FUNCTION_BLOCK AI_1_Module
VAR
	{attribute addProperty Name  "1"}
	iCHANNEL_1 : AI_Channel;
	{attribute addProperty Name  "WcState"}
	WcState : WcState;
	{attribute addProperty Name  "WcState"}
	InfoData : WcState;
END_VAR

END_FUNCTION_BLOCK

(* stored: Version 1.1.0.1, ProductVersion 3.1.4024.6
   POU AI_1_Module: Id {18690fd6-f1b5-4e14-bdd5-5776974196f1}, SpecialFunc None *)
